// TIA Portal V19 export
DATA_BLOCK "DB_GroupConfig"   // DB42
{ S7_Optimized_Access := 'FALSE' }
// stored: AutoNumber false
   VAR RETAIN
      AnzGroup : Int := 0;   // + Anzahl der Definierten Gruppen (wird mit FW-Editor eingetragen)
      OffsetAdr : Int := 10;   // * Adresse der ersten Gruppendefinition
      resW : Int := 0;
      resD1 : DInt := 0;
      Gruppe : Array[0..9] of Struct   // * Feldlänge anpassen (Inhalte werden mit FW-Editor erzeugt)
         Start : Int;   // + Startadresse in Byte der Gruppe in diesem DB sieh Def
         QT_Nr : Int;   // + zu benutzender Quertransport, wenn reihenübergreifende Gruppe
         Skip_enable : Bool;   // + Überspringen möglich
         OptiGroup : Bool;   // + Optimierungsberechnung berücksichtigen
         Vorzugsreihe : Bool;   // + Vorzugsweise innerhalb der gleichen Reihe umsetzen
         res3 : Bool;
         res4 : Bool;
         res5 : Bool;
         res6 : Bool;
         res7 : Bool;
         res8 : Bool;
         res9 : Bool;
         res10 : Bool;
         res11 : Bool;
         res12 : Bool;
         res13 : Bool;
         res14 : Bool;
         res15 : Bool;
      END_STRUCT;
      Def : Array[1..10] of Byte;   // * Definition der Gruppen-Positionen
   END_VAR
BEGIN
   Gruppe[0..9].Start := 0;
   Gruppe[0..9].QT_Nr := 0;
   Gruppe[0..9].Skip_enable := FALSE;
   Gruppe[0..9].OptiGroup := FALSE;
   Gruppe[0..9].Vorzugsreihe := FALSE;
   Gruppe[0..9].res3 := FALSE;
   Gruppe[0..9].res4 := FALSE;
   Gruppe[0..9].res5 := FALSE;
   Gruppe[0..9].res6 := FALSE;
   Gruppe[0..9].res7 := FALSE;
   Gruppe[0..9].res8 := FALSE;
   Gruppe[0..9].res9 := FALSE;
   Gruppe[0..9].res10 := FALSE;
   Gruppe[0..9].res11 := FALSE;
   Gruppe[0..9].res12 := FALSE;
   Gruppe[0..9].res13 := FALSE;
   Gruppe[0..9].res14 := FALSE;
   Gruppe[0..9].res15 := FALSE;
   Def[1..10] := 16#00;
END_DATA_BLOCK
